PROGRAM P_Demo_F_YearIsLeapYear
VAR
    wYear       : WORD := 2024; // 要判断的年份
    bIsLeapYear : BOOL; // TRUE = 闰年
    bRunOnce    : BOOL; // 脉冲触发
END_VAR

// =============================================================================
// 场景：HMI 让用户输入日期时需校验 2 月 29 日是否合法
//
// 价值：1 行调用避免手写 100/400 三段判定，最容易漏的是「能被 100 整除但不被 400 整除非闰年」
//
// 验证步骤：
//   1. 引用 Tc2_Utilities
//   2. 编译 + 登录 + 运行
//   3. 强制 bRunOnce := TRUE
//   4. 在线观察 bIsLeapYear = TRUE（2024 是闰年）
//   5. wYear:=1900 → FALSE（100 整除但 400 不整除）
//   6. wYear:=2000 → TRUE（400 整除）
// =============================================================================
bIsLeapYear := F_YearIsLeapYear(wYear);

END_PROGRAM

(* stored: Version 1.1.0.1, ProductVersion 3.1.4024.5
   POU P_Demo_F_YearIsLeapYear: Id {4af73ee2-e2d4-5e8d-ad9d-74e3b52d04e1}, SpecialFunc None *)
